{attribute 'qualified_only'}
VAR_GLOBAL
END_VAR

(* stored: Version 1.1.0.1, ProductVersion 3.1.4022.7
   GVL GVL_01_Shift: Id {61893bdd-dafd-4483-b68b-ed23fdbc25e4} *)
